PROGRAM POU
VAR
END_VAR

END_PROGRAM

(* stored: Version 1.1.0.1, ProductVersion 3.1.4024.0
   POU POU: Id {19167c9e-9ce1-4b37-93f1-33aedbe2aeb9}, SpecialFunc None *)
